DATA_BLOCK "DB_Commissioning"
{ S7_Optimized_Access := 'TRUE' }
VERSION : 0.1
NON_RETAIN
// ATTRIBUTES
// AUTO_NUMBER = False
// BLOCK_NUMBER = 32767
// END_ATTRIBUTES
   VAR RETAIN
      str : Array[1..8] of String[60];
      bit : Array[1..8] of Bool;
   END_VAR


BEGIN
   str[1] := 'LE4B171420124M33700000131950710';

END_DATA_BLOCK

